{attribute 'GeneratedUsingTerminal: EL2212-0000-0020'}
{attribute addProperty BoxType "EL2212-0000-0020"}
{attribute addProperty Id "OutputBOOL1TristateBOOL1PWMBOOL1ResetBOOL1"}
{attribute addProperty CRC "2266459167"}
{attribute addProperty Size "4"}
TYPE Control_87176C1F :
STRUCT
	{attribute addProperty Name "Output"}
	Output : BOOL;
	{attribute addProperty Name "Tristate"}
	Tristate : BOOL;
	{attribute addProperty Name "PWM"}
	PWM : BOOL;
	{attribute addProperty Name "Reset"}
	Reset : BOOL;
END_STRUCT
END_TYPE

(* stored: Version 1.2.0.0, ProductVersion 3.1.4024.9
   DUT Control_87176C1F: Id {d79601e6-dfb8-4aa5-9e56-54aaec1b011a} *)
